{attribute addProperty BoxType "APS1003-7000-0016"}
{attribute addProperty Id "YVR_InputsAT %I*YVR_Inputs_32B3017D784980YVR_OutputsAT %Q*YVR_Outputs_0CD1622111681460WcStateAT %I*WcState_F855686C1620InfoDataAT %I*InfoData_0BDED7BF144180"}
{attribute addProperty CRC "128310746"}
{attribute addProperty SizeInBites "2112"}
{attribute addProperty SizeInBytes "264"}
TYPE APS1003_C39F7B89 :
STRUCT
	{attribute addProperty Name "YVR_Inputs"}
	YVR_Inputs : YVR_Inputs_32B3017D;
	{attribute addProperty Name "YVR_Outputs"}
	YVR_Outputs : YVR_Outputs_0CD16221;
	{attribute addProperty Name "WcState"}
	WcState : WcState_F855686C;
	{attribute addProperty Name "InfoData"}
	InfoData : InfoData_0BDED7BF;
END_STRUCT
END_TYPE

(* stored: Version 1.2.0.0, ProductVersion 3.1.4024.9
   DUT APS1003_C39F7B89: Id {1de2d034-6a13-458d-acff-3fdfaeabe7fc} *)
